FUNCTION_BLOCK HazardTimer
VAR_INPUT
	bTriggH: BOOL;
	bINH: BOOL;
END_VAR
VAR_OUTPUT
	tTimeH: TIME;
	bQH: BOOL;
END_VAR
VAR
	tTimerH: ton;
END_VAR

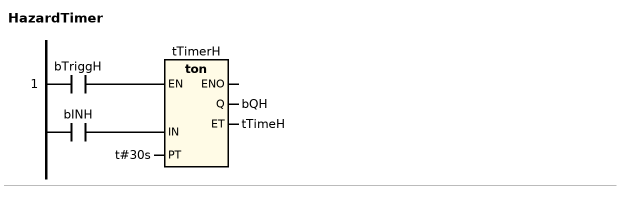
// NETWORK 1
IF bTriggH THEN
    tTimerH(IN := bINH, PT := t#30s, Q => bQH, ET => tTimeH); // ton
END_IF

END_FUNCTION_BLOCK

(* stored: Version 1.1.0.1, ProductVersion 3.1.4018.9
   POU HazardTimer: Id {e14c892d-f1f8-42c7-8a90-9e0244fb9f56}, SpecialFunc None *)
